# EPICS substitutions: iocAdminLib/Db/iocSoft.substitutions
#==============================================================================
#
# Abs:  IOC Administration Records
#
# Name: iocSoft.substitutions
#
#==============================================================================
#
file iocSoft.template
{
	pattern
	{ IOCNAME }
	{ $(IOC)  }
}

file iocEnvVars.db
{
	pattern
	{ IOCNAME }
	{ $(IOC)  }
}
